TYPE St_DataHisto_Epoch :
STRUCT
	Timestamp		: ULINT;
	ParentId		: DINT;
	Value			: LREAL;
END_STRUCT
END_TYPE

(* stored: Version 1.1.0.1, ProductVersion 3.1.4024.6
   DUT St_DataHisto_Epoch: Id {3782bbbd-b4d8-4652-86bc-36492ee5e372} *)
